PROGRAM P00_OP
VAR		
	N_OP_CMD AT%MB64:  ARRAY [0..35] OF BYTE;//op cmd 주소
	memSetResult: UDINT;	
	b_Test: BOOL;
END_VAR
VAR // added by the converter: edge detectors and wires of the graphical bodies
    _rt1, _rt2, _rt3, _rt4, _rt5, _rt6, _rt7, _rt8, _rt9, _rt10, _rt11, _rt12, _rt13, _rt14, _rt15, _rt16, _rt17, _rt18, _rt19, _rt20, _rt21, _rt22, _rt23, _rt24, _rt25, _rt26, _rt27, _rt28, _rt29, _rt30, _rt31, _rt32, _rt33, _rt34, _rt35, _rt36, _rt37, _rt38, _rt39, _rt40, _rt41, _rt42, _rt43, _rt44, _rt45, _rt46, _rt47, _rt48, _rt49, _rt50, _rt51, _rt52, _rt53, _rt54, _rt55, _rt56, _rt57, _rt58, _rt59, _rt60, _rt61, _rt62, _rt63, _rt64, _rt65, _rt66, _rt67, _rt68, _rt69, _rt70, _rt71, _rt72, _rt73, _rt74, _rt75, _rt76, _rt77, _rt78, _rt79, _rt80, _rt81, _rt82, _rt83, _rt84, _rt85, _rt86, _rt87, _rt88, _rt89, _rt90, _rt91, _rt92, _rt93, _rt94, _rt95, _rt96, _rt97, _rt98, _rt99, _rt100, _rt101, _rt102, _rt103, _rt104, _rt105, _rt106, _rt107, _rt108, _rt109, _rt110, _rt111, _rt112, _rt113, _rt114, _rt115, _rt116, _rt117, _rt118, _rt119, _rt120, _rt121, _rt122, _rt123, _rt124, _rt125, _rt126, _rt127, _rt128, _rt129, _rt130, _rt131, _rt132, _rt133, _rt134, _rt135, _rt136, _rt137, _rt138, _rt139, _rt140, _rt141, _rt142, _rt143, _rt144, _rt145, _rt146, _rt147, _rt148, _rt149, _rt150, _rt151, _rt152, _rt153, _rt154, _rt155, _rt156, _rt157, _rt158, _rt159, _rt160, _rt161, _rt162, _rt163, _rt164, _rt165, _rt166, _rt167, _rt168, _rt169, _rt170, _rt171, _rt172, _rt173, _rt174, _rt175, _rt176, _rt177, _rt178, _rt179, _rt180, _rt181, _rt182, _rt183, _rt184, _rt185, _rt186, _rt187, _rt188, _rt189, _rt190, _rt191, _rt192, _rt193, _rt194, _rt195, _rt196, _rt197, _rt198, _rt199, _rt200, _rt201, _rt202, _rt203, _rt204, _rt205, _rt206, _rt207, _rt208, _rt209, _rt210, _rt211, _rt212, _rt213, _rt214, _rt215, _rt216, _rt217, _rt218, _rt219, _rt220, _rt221, _rt222, _rt223, _rt224, _rt225, _rt226, _rt227, _rt228, _rt229, _rt230, _rt231, _rt232, _rt233, _rt234 : R_TRIG;
    _w1, _w2, _w3, _w4, _w5, _w6, _w7, _w8, _w9, _w10, _w11, _w12 : BOOL;
END_VAR

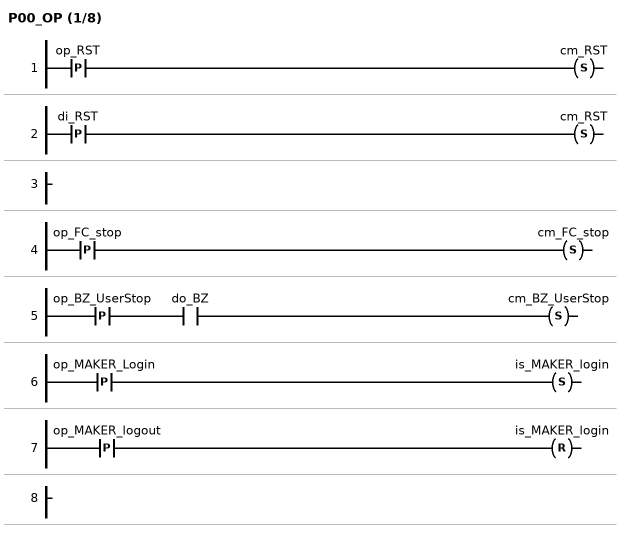
// NETWORK 1
_rt1(CLK := op_RST);
cm_RST S= _rt1.Q;

// NETWORK 2
_rt2(CLK := di_RST);
cm_RST S= _rt2.Q;

// NETWORK 3

// NETWORK 4
_rt3(CLK := op_FC_stop);
cm_FC_stop S= _rt3.Q;

// NETWORK 5
_rt4(CLK := op_BZ_UserStop);
cm_BZ_UserStop S= _rt4.Q AND do_BZ;

// NETWORK 6
_rt5(CLK := op_MAKER_Login);
is_MAKER_login S= _rt5.Q;

// NETWORK 7
_rt6(CLK := op_MAKER_logout);
is_MAKER_login R= _rt6.Q;

// NETWORK 8

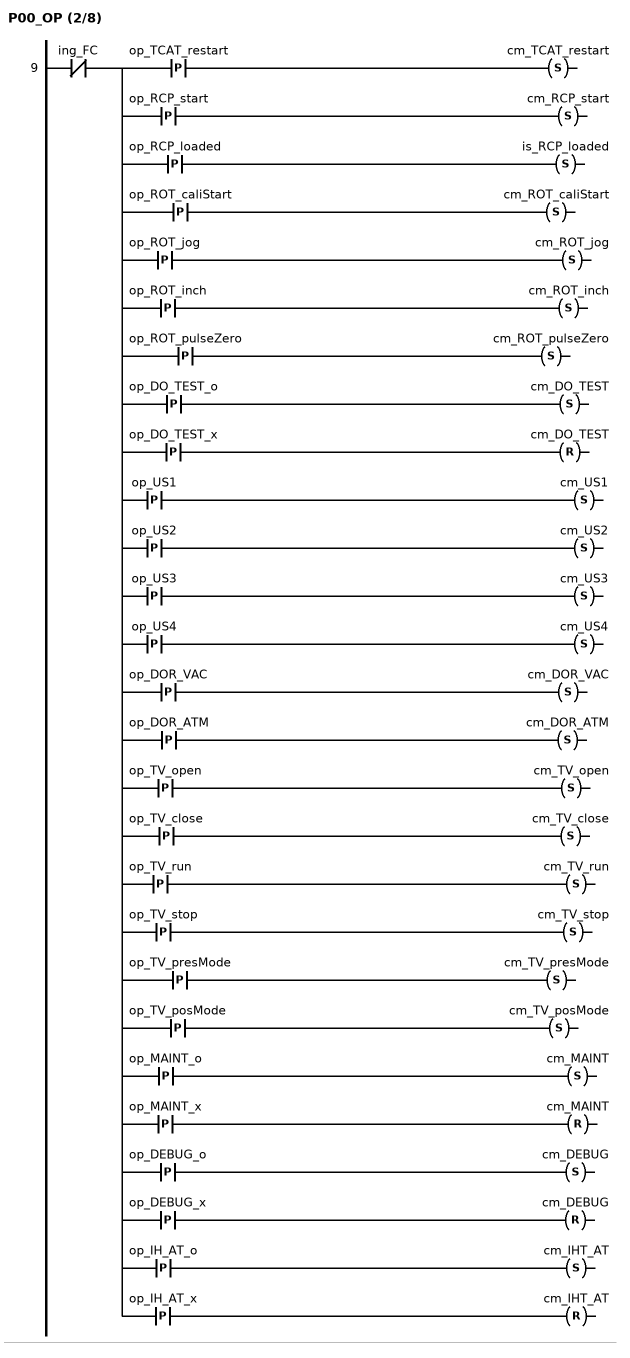
// NETWORK 9
_w1 := NOT ing_FC;
_rt7(CLK := op_TCAT_restart);
cm_TCAT_restart S= _w1 AND _rt7.Q;
_rt8(CLK := op_RCP_start);
cm_RCP_start S= _w1 AND _rt8.Q;
_rt9(CLK := op_RCP_loaded);
is_RCP_loaded S= _w1 AND _rt9.Q;
_rt10(CLK := op_ROT_caliStart);
cm_ROT_caliStart S= _w1 AND _rt10.Q;
_rt11(CLK := op_ROT_jog);
cm_ROT_jog S= _w1 AND _rt11.Q;
_rt12(CLK := op_ROT_inch);
cm_ROT_inch S= _w1 AND _rt12.Q;
_rt13(CLK := op_ROT_pulseZero);
cm_ROT_pulseZero S= _w1 AND _rt13.Q;
_rt14(CLK := op_DO_TEST_o);
cm_DO_TEST S= _w1 AND _rt14.Q;
_rt15(CLK := op_DO_TEST_x);
cm_DO_TEST R= _w1 AND _rt15.Q;
_rt16(CLK := op_US1);
cm_US1 S= _w1 AND _rt16.Q;
_rt17(CLK := op_US2);
cm_US2 S= _w1 AND _rt17.Q;
_rt18(CLK := op_US3);
cm_US3 S= _w1 AND _rt18.Q;
_rt19(CLK := op_US4);
cm_US4 S= _w1 AND _rt19.Q;
_rt20(CLK := op_DOR_VAC);
cm_DOR_VAC S= _w1 AND _rt20.Q;
_rt21(CLK := op_DOR_ATM);
cm_DOR_ATM S= _w1 AND _rt21.Q;
_rt22(CLK := op_TV_open);
cm_TV_open S= _w1 AND _rt22.Q;
_rt23(CLK := op_TV_close);
cm_TV_close S= _w1 AND _rt23.Q;
_rt24(CLK := op_TV_run);
cm_TV_run S= _w1 AND _rt24.Q;
_rt25(CLK := op_TV_stop);
cm_TV_stop S= _w1 AND _rt25.Q;
_rt26(CLK := op_TV_presMode);
cm_TV_presMode S= _w1 AND _rt26.Q;
_rt27(CLK := op_TV_posMode);
cm_TV_posMode S= _w1 AND _rt27.Q;
_rt28(CLK := op_MAINT_o);
cm_MAINT S= _w1 AND _rt28.Q;
_rt29(CLK := op_MAINT_x);
cm_MAINT R= _w1 AND _rt29.Q;
_rt30(CLK := op_DEBUG_o);
cm_DEBUG S= _w1 AND _rt30.Q;
_rt31(CLK := op_DEBUG_x);
cm_DEBUG R= _w1 AND _rt31.Q;
_rt32(CLK := op_IH_AT_o);
cm_IHT_AT S= _w1 AND _rt32.Q;
_rt33(CLK := op_IH_AT_x);
cm_IHT_AT R= _w1 AND _rt33.Q;

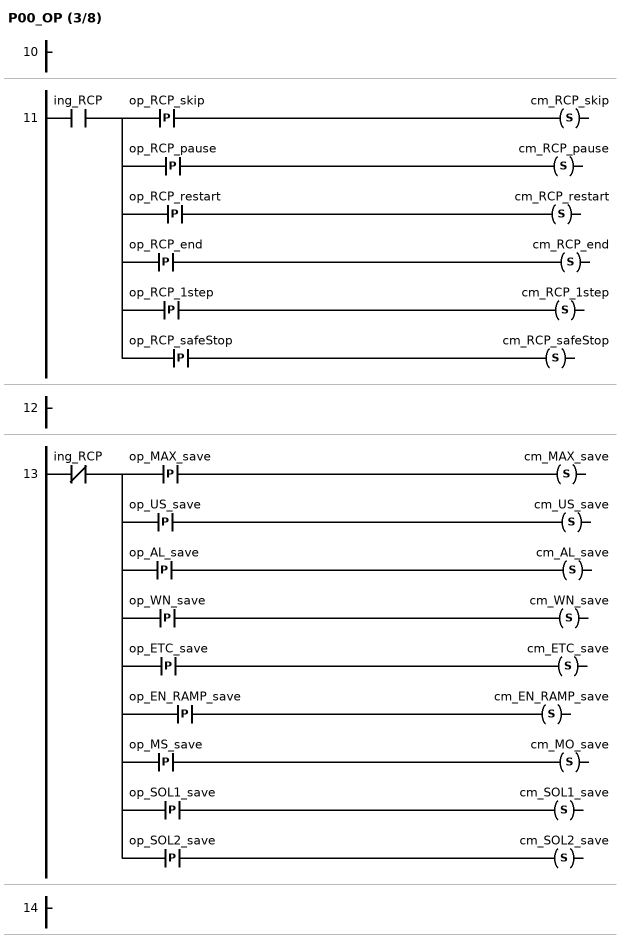
// NETWORK 10

// NETWORK 11
_rt34(CLK := op_RCP_skip);
cm_RCP_skip S= ing_RCP AND _rt34.Q;
_rt35(CLK := op_RCP_pause);
cm_RCP_pause S= ing_RCP AND _rt35.Q;
_rt36(CLK := op_RCP_restart);
cm_RCP_restart S= ing_RCP AND _rt36.Q;
_rt37(CLK := op_RCP_end);
cm_RCP_end S= ing_RCP AND _rt37.Q;
_rt38(CLK := op_RCP_1step);
cm_RCP_1step S= ing_RCP AND _rt38.Q;
_rt39(CLK := op_RCP_safeStop);
cm_RCP_safeStop S= ing_RCP AND _rt39.Q;

// NETWORK 12

// NETWORK 13
_w2 := NOT ing_RCP;
_rt40(CLK := op_MAX_save);
cm_MAX_save S= _w2 AND _rt40.Q;
_rt41(CLK := op_US_save);
cm_US_save S= _w2 AND _rt41.Q;
_rt42(CLK := op_AL_save);
cm_AL_save S= _w2 AND _rt42.Q;
_rt43(CLK := op_WN_save);
cm_WN_save S= _w2 AND _rt43.Q;
_rt44(CLK := op_ETC_save);
cm_ETC_save S= _w2 AND _rt44.Q;
_rt45(CLK := op_EN_RAMP_save);
cm_EN_RAMP_save S= _w2 AND _rt45.Q;
_rt46(CLK := op_MS_save);
cm_MO_save S= _w2 AND _rt46.Q;
_rt47(CLK := op_SOL1_save);
cm_SOL1_save S= _w2 AND _rt47.Q;
_rt48(CLK := op_SOL2_save);
cm_SOL2_save S= _w2 AND _rt48.Q;

// NETWORK 14

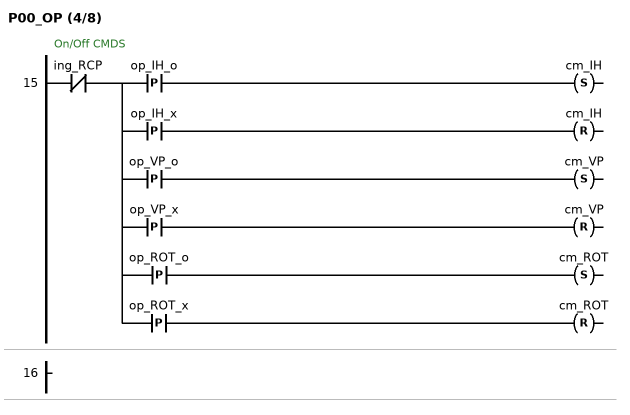
// NETWORK 15
// On/Off CMDS
_w3 := NOT ing_RCP;
_rt49(CLK := op_IH_o);
cm_IH S= _w3 AND _rt49.Q;
_rt50(CLK := op_IH_x);
cm_IH R= _w3 AND _rt50.Q;
_rt51(CLK := op_VP_o);
cm_VP S= _w3 AND _rt51.Q;
_rt52(CLK := op_VP_x);
cm_VP R= _w3 AND _rt52.Q;
_rt53(CLK := op_ROT_o);
cm_ROT S= _w3 AND _rt53.Q;
_rt54(CLK := op_ROT_x);
cm_ROT R= _w3 AND _rt54.Q;

// NETWORK 16

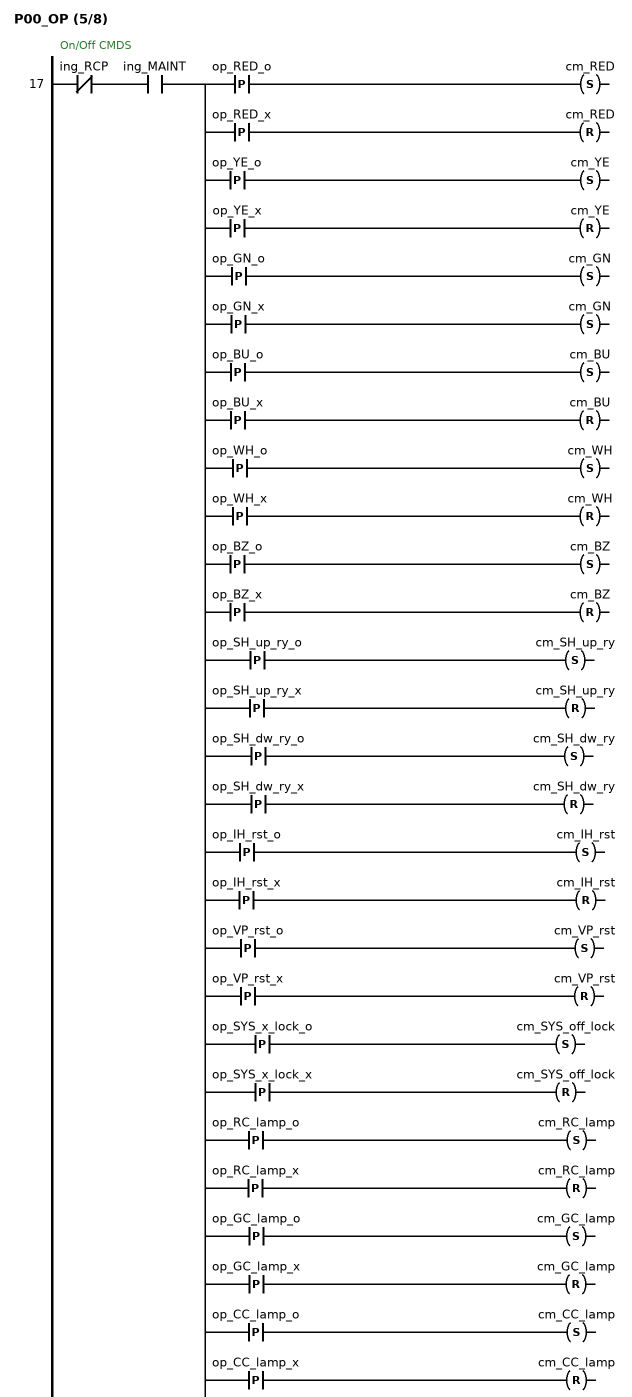
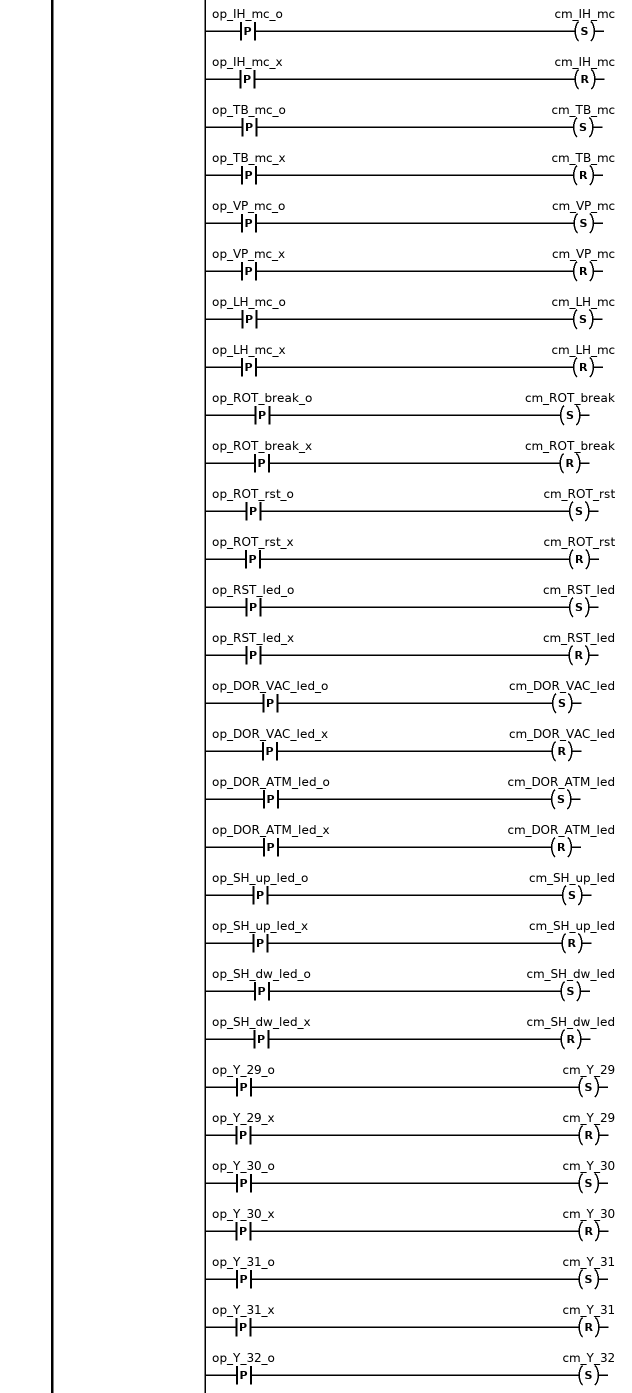
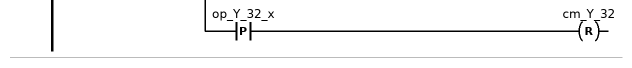
// NETWORK 17
// On/Off CMDS
_w4 := NOT ing_RCP AND ing_MAINT;
_rt55(CLK := op_RED_o);
cm_RED S= _w4 AND _rt55.Q;
_rt56(CLK := op_RED_x);
cm_RED R= _w4 AND _rt56.Q;
_rt57(CLK := op_YE_o);
cm_YE S= _w4 AND _rt57.Q;
_rt58(CLK := op_YE_x);
cm_YE R= _w4 AND _rt58.Q;
_rt59(CLK := op_GN_o);
cm_GN S= _w4 AND _rt59.Q;
_rt60(CLK := op_GN_x);
cm_GN S= _w4 AND _rt60.Q;
_rt61(CLK := op_BU_o);
cm_BU S= _w4 AND _rt61.Q;
_rt62(CLK := op_BU_x);
cm_BU R= _w4 AND _rt62.Q;
_rt63(CLK := op_WH_o);
cm_WH S= _w4 AND _rt63.Q;
_rt64(CLK := op_WH_x);
cm_WH R= _w4 AND _rt64.Q;
_rt65(CLK := op_BZ_o);
cm_BZ S= _w4 AND _rt65.Q;
_rt66(CLK := op_BZ_x);
cm_BZ R= _w4 AND _rt66.Q;
_rt67(CLK := op_SH_up_ry_o);
cm_SH_up_ry S= _w4 AND _rt67.Q;
_rt68(CLK := op_SH_up_ry_x);
cm_SH_up_ry R= _w4 AND _rt68.Q;
_rt69(CLK := op_SH_dw_ry_o);
cm_SH_dw_ry S= _w4 AND _rt69.Q;
_rt70(CLK := op_SH_dw_ry_x);
cm_SH_dw_ry R= _w4 AND _rt70.Q;
_rt71(CLK := op_IH_rst_o);
cm_IH_rst S= _w4 AND _rt71.Q;
_rt72(CLK := op_IH_rst_x);
cm_IH_rst R= _w4 AND _rt72.Q;
_rt73(CLK := op_VP_rst_o);
cm_VP_rst S= _w4 AND _rt73.Q;
_rt74(CLK := op_VP_rst_x);
cm_VP_rst R= _w4 AND _rt74.Q;
_rt75(CLK := op_SYS_x_lock_o);
cm_SYS_off_lock S= _w4 AND _rt75.Q;
_rt76(CLK := op_SYS_x_lock_x);
cm_SYS_off_lock R= _w4 AND _rt76.Q;
_rt77(CLK := op_RC_lamp_o);
cm_RC_lamp S= _w4 AND _rt77.Q;
_rt78(CLK := op_RC_lamp_x);
cm_RC_lamp R= _w4 AND _rt78.Q;
_rt79(CLK := op_GC_lamp_o);
cm_GC_lamp S= _w4 AND _rt79.Q;
_rt80(CLK := op_GC_lamp_x);
cm_GC_lamp R= _w4 AND _rt80.Q;
_rt81(CLK := op_CC_lamp_o);
cm_CC_lamp S= _w4 AND _rt81.Q;
_rt82(CLK := op_CC_lamp_x);
cm_CC_lamp R= _w4 AND _rt82.Q;
_rt83(CLK := op_IH_mc_o);
cm_IH_mc S= _w4 AND _rt83.Q;
_rt84(CLK := op_IH_mc_x);
cm_IH_mc R= _w4 AND _rt84.Q;
_rt85(CLK := op_TB_mc_o);
cm_TB_mc S= _w4 AND _rt85.Q;
_rt86(CLK := op_TB_mc_x);
cm_TB_mc R= _w4 AND _rt86.Q;
_rt87(CLK := op_VP_mc_o);
cm_VP_mc S= _w4 AND _rt87.Q;
_rt88(CLK := op_VP_mc_x);
cm_VP_mc R= _w4 AND _rt88.Q;
_rt89(CLK := op_LH_mc_o);
cm_LH_mc S= _w4 AND _rt89.Q;
_rt90(CLK := op_LH_mc_x);
cm_LH_mc R= _w4 AND _rt90.Q;
_rt91(CLK := op_ROT_break_o);
cm_ROT_break S= _w4 AND _rt91.Q;
_rt92(CLK := op_ROT_break_x);
cm_ROT_break R= _w4 AND _rt92.Q;
_rt93(CLK := op_ROT_rst_o);
cm_ROT_rst S= _w4 AND _rt93.Q;
_rt94(CLK := op_ROT_rst_x);
cm_ROT_rst R= _w4 AND _rt94.Q;
_rt95(CLK := op_RST_led_o);
cm_RST_led S= _w4 AND _rt95.Q;
_rt96(CLK := op_RST_led_x);
cm_RST_led R= _w4 AND _rt96.Q;
_rt97(CLK := op_DOR_VAC_led_o);
cm_DOR_VAC_led S= _w4 AND _rt97.Q;
_rt98(CLK := op_DOR_VAC_led_x);
cm_DOR_VAC_led R= _w4 AND _rt98.Q;
_rt99(CLK := op_DOR_ATM_led_o);
cm_DOR_ATM_led S= _w4 AND _rt99.Q;
_rt100(CLK := op_DOR_ATM_led_x);
cm_DOR_ATM_led R= _w4 AND _rt100.Q;
_rt101(CLK := op_SH_up_led_o);
cm_SH_up_led S= _w4 AND _rt101.Q;
_rt102(CLK := op_SH_up_led_x);
cm_SH_up_led R= _w4 AND _rt102.Q;
_rt103(CLK := op_SH_dw_led_o);
cm_SH_dw_led S= _w4 AND _rt103.Q;
_rt104(CLK := op_SH_dw_led_x);
cm_SH_dw_led R= _w4 AND _rt104.Q;
_rt105(CLK := op_Y_29_o);
cm_Y_29 S= _w4 AND _rt105.Q;
_rt106(CLK := op_Y_29_x);
cm_Y_29 R= _w4 AND _rt106.Q;
_rt107(CLK := op_Y_30_o);
cm_Y_30 S= _w4 AND _rt107.Q;
_rt108(CLK := op_Y_30_x);
cm_Y_30 R= _w4 AND _rt108.Q;
_rt109(CLK := op_Y_31_o);
cm_Y_31 S= _w4 AND _rt109.Q;
_rt110(CLK := op_Y_31_x);
cm_Y_31 R= _w4 AND _rt110.Q;
_rt111(CLK := op_Y_32_o);
cm_Y_32 S= _w4 AND _rt111.Q;
_rt112(CLK := op_Y_32_x);
cm_Y_32 R= _w4 AND _rt112.Q;

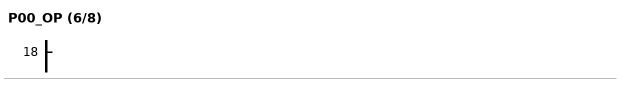
// NETWORK 18

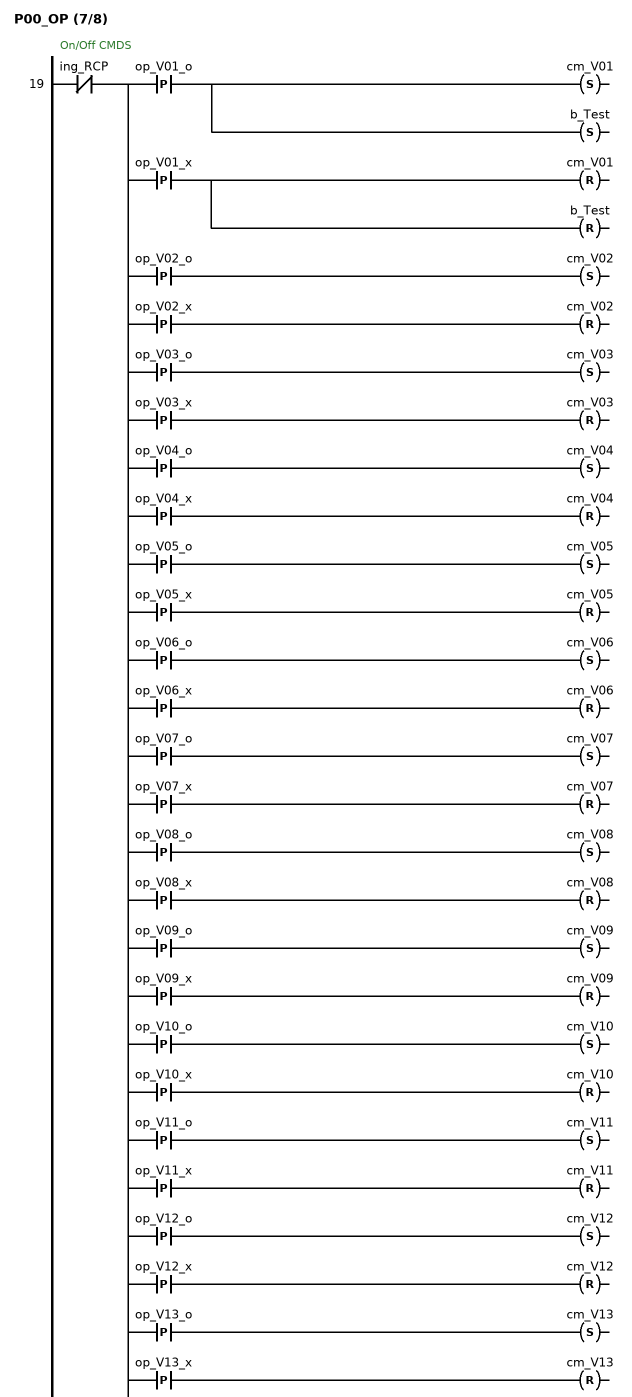
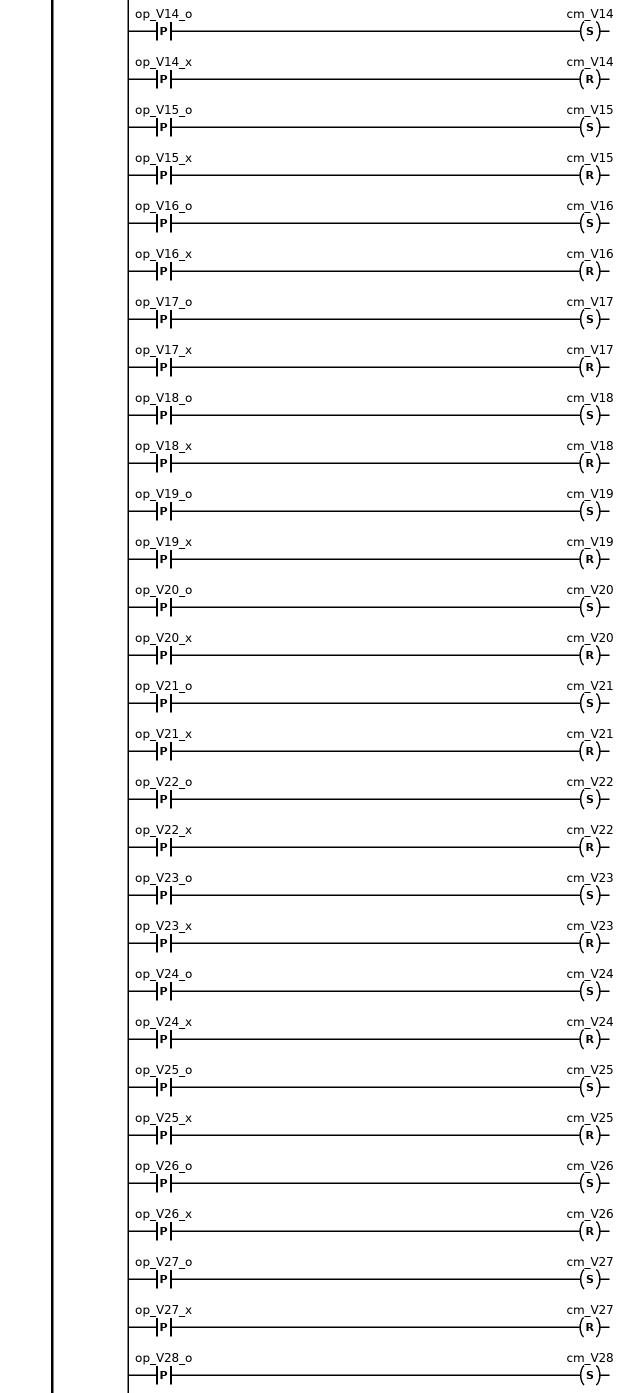
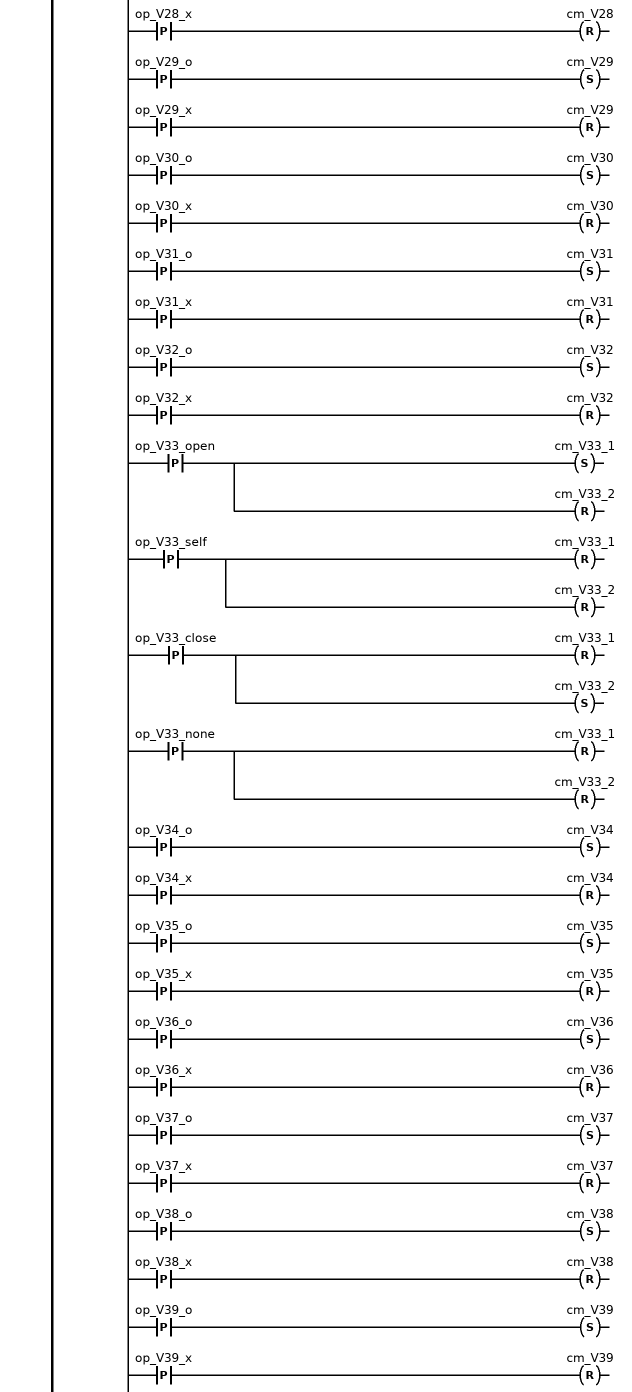
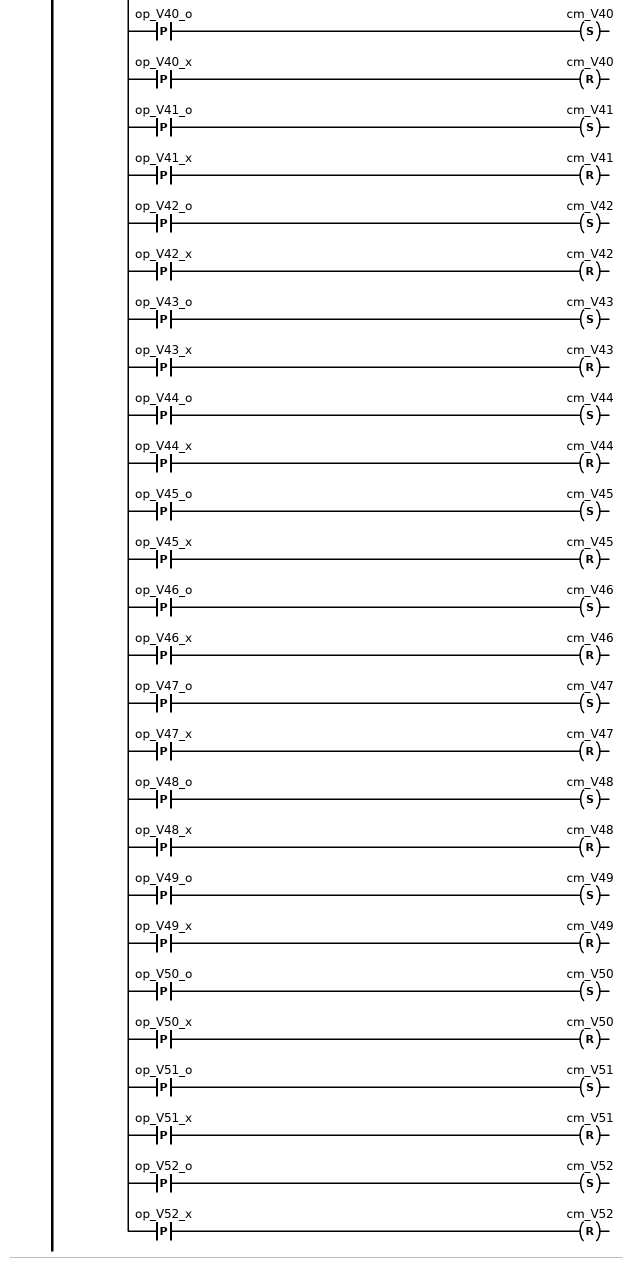
// NETWORK 19
// On/Off CMDS
_w5 := NOT ing_RCP;
_rt113(CLK := op_V01_o);
_w6 := _w5 AND _rt113.Q;
cm_V01 S= _w6;
b_Test S= _w6;
_rt114(CLK := op_V01_x);
_w7 := _w5 AND _rt114.Q;
cm_V01 R= _w7;
b_Test R= _w7;
_rt115(CLK := op_V02_o);
cm_V02 S= _w5 AND _rt115.Q;
_rt116(CLK := op_V02_x);
cm_V02 R= _w5 AND _rt116.Q;
_rt117(CLK := op_V03_o);
cm_V03 S= _w5 AND _rt117.Q;
_rt118(CLK := op_V03_x);
cm_V03 R= _w5 AND _rt118.Q;
_rt119(CLK := op_V04_o);
cm_V04 S= _w5 AND _rt119.Q;
_rt120(CLK := op_V04_x);
cm_V04 R= _w5 AND _rt120.Q;
_rt121(CLK := op_V05_o);
cm_V05 S= _w5 AND _rt121.Q;
_rt122(CLK := op_V05_x);
cm_V05 R= _w5 AND _rt122.Q;
_rt123(CLK := op_V06_o);
cm_V06 S= _w5 AND _rt123.Q;
_rt124(CLK := op_V06_x);
cm_V06 R= _w5 AND _rt124.Q;
_rt125(CLK := op_V07_o);
cm_V07 S= _w5 AND _rt125.Q;
_rt126(CLK := op_V07_x);
cm_V07 R= _w5 AND _rt126.Q;
_rt127(CLK := op_V08_o);
cm_V08 S= _w5 AND _rt127.Q;
_rt128(CLK := op_V08_x);
cm_V08 R= _w5 AND _rt128.Q;
_rt129(CLK := op_V09_o);
cm_V09 S= _w5 AND _rt129.Q;
_rt130(CLK := op_V09_x);
cm_V09 R= _w5 AND _rt130.Q;
_rt131(CLK := op_V10_o);
cm_V10 S= _w5 AND _rt131.Q;
_rt132(CLK := op_V10_x);
cm_V10 R= _w5 AND _rt132.Q;
_rt133(CLK := op_V11_o);
cm_V11 S= _w5 AND _rt133.Q;
_rt134(CLK := op_V11_x);
cm_V11 R= _w5 AND _rt134.Q;
_rt135(CLK := op_V12_o);
cm_V12 S= _w5 AND _rt135.Q;
_rt136(CLK := op_V12_x);
cm_V12 R= _w5 AND _rt136.Q;
_rt137(CLK := op_V13_o);
cm_V13 S= _w5 AND _rt137.Q;
_rt138(CLK := op_V13_x);
cm_V13 R= _w5 AND _rt138.Q;
_rt139(CLK := op_V14_o);
cm_V14 S= _w5 AND _rt139.Q;
_rt140(CLK := op_V14_x);
cm_V14 R= _w5 AND _rt140.Q;
_rt141(CLK := op_V15_o);
cm_V15 S= _w5 AND _rt141.Q;
_rt142(CLK := op_V15_x);
cm_V15 R= _w5 AND _rt142.Q;
_rt143(CLK := op_V16_o);
cm_V16 S= _w5 AND _rt143.Q;
_rt144(CLK := op_V16_x);
cm_V16 R= _w5 AND _rt144.Q;
_rt145(CLK := op_V17_o);
cm_V17 S= _w5 AND _rt145.Q;
_rt146(CLK := op_V17_x);
cm_V17 R= _w5 AND _rt146.Q;
_rt147(CLK := op_V18_o);
cm_V18 S= _w5 AND _rt147.Q;
_rt148(CLK := op_V18_x);
cm_V18 R= _w5 AND _rt148.Q;
_rt149(CLK := op_V19_o);
cm_V19 S= _w5 AND _rt149.Q;
_rt150(CLK := op_V19_x);
cm_V19 R= _w5 AND _rt150.Q;
_rt151(CLK := op_V20_o);
cm_V20 S= _w5 AND _rt151.Q;
_rt152(CLK := op_V20_x);
cm_V20 R= _w5 AND _rt152.Q;
_rt153(CLK := op_V21_o);
cm_V21 S= _w5 AND _rt153.Q;
_rt154(CLK := op_V21_x);
cm_V21 R= _w5 AND _rt154.Q;
_rt155(CLK := op_V22_o);
cm_V22 S= _w5 AND _rt155.Q;
_rt156(CLK := op_V22_x);
cm_V22 R= _w5 AND _rt156.Q;
_rt157(CLK := op_V23_o);
cm_V23 S= _w5 AND _rt157.Q;
_rt158(CLK := op_V23_x);
cm_V23 R= _w5 AND _rt158.Q;
_rt159(CLK := op_V24_o);
cm_V24 S= _w5 AND _rt159.Q;
_rt160(CLK := op_V24_x);
cm_V24 R= _w5 AND _rt160.Q;
_rt161(CLK := op_V25_o);
cm_V25 S= _w5 AND _rt161.Q;
_rt162(CLK := op_V25_x);
cm_V25 R= _w5 AND _rt162.Q;
_rt163(CLK := op_V26_o);
cm_V26 S= _w5 AND _rt163.Q;
_rt164(CLK := op_V26_x);
cm_V26 R= _w5 AND _rt164.Q;
_rt165(CLK := op_V27_o);
cm_V27 S= _w5 AND _rt165.Q;
_rt166(CLK := op_V27_x);
cm_V27 R= _w5 AND _rt166.Q;
_rt167(CLK := op_V28_o);
cm_V28 S= _w5 AND _rt167.Q;
_rt168(CLK := op_V28_x);
cm_V28 R= _w5 AND _rt168.Q;
_rt169(CLK := op_V29_o);
cm_V29 S= _w5 AND _rt169.Q;
_rt170(CLK := op_V29_x);
cm_V29 R= _w5 AND _rt170.Q;
_rt171(CLK := op_V30_o);
cm_V30 S= _w5 AND _rt171.Q;
_rt172(CLK := op_V30_x);
cm_V30 R= _w5 AND _rt172.Q;
_rt173(CLK := op_V31_o);
cm_V31 S= _w5 AND _rt173.Q;
_rt174(CLK := op_V31_x);
cm_V31 R= _w5 AND _rt174.Q;
_rt175(CLK := op_V32_o);
cm_V32 S= _w5 AND _rt175.Q;
_rt176(CLK := op_V32_x);
cm_V32 R= _w5 AND _rt176.Q;
_rt177(CLK := op_V33_open);
_w8 := _w5 AND _rt177.Q;
cm_V33_1 S= _w8;
cm_V33_2 R= _w8;
_rt178(CLK := op_V33_self);
_w9 := _w5 AND _rt178.Q;
cm_V33_1 R= _w9;
cm_V33_2 R= _w9;
_rt179(CLK := op_V33_close);
_w10 := _w5 AND _rt179.Q;
cm_V33_1 R= _w10;
cm_V33_2 S= _w10;
_rt180(CLK := op_V33_none);
_w11 := _w5 AND _rt180.Q;
cm_V33_1 R= _w11;
cm_V33_2 R= _w11;
_rt181(CLK := op_V34_o);
cm_V34 S= _w5 AND _rt181.Q;
_rt182(CLK := op_V34_x);
cm_V34 R= _w5 AND _rt182.Q;
_rt183(CLK := op_V35_o);
cm_V35 S= _w5 AND _rt183.Q;
_rt184(CLK := op_V35_x);
cm_V35 R= _w5 AND _rt184.Q;
_rt185(CLK := op_V36_o);
cm_V36 S= _w5 AND _rt185.Q;
_rt186(CLK := op_V36_x);
cm_V36 R= _w5 AND _rt186.Q;
_rt187(CLK := op_V37_o);
cm_V37 S= _w5 AND _rt187.Q;
_rt188(CLK := op_V37_x);
cm_V37 R= _w5 AND _rt188.Q;
_rt189(CLK := op_V38_o);
cm_V38 S= _w5 AND _rt189.Q;
_rt190(CLK := op_V38_x);
cm_V38 R= _w5 AND _rt190.Q;
_rt191(CLK := op_V39_o);
cm_V39 S= _w5 AND _rt191.Q;
_rt192(CLK := op_V39_x);
cm_V39 R= _w5 AND _rt192.Q;
_rt193(CLK := op_V40_o);
cm_V40 S= _w5 AND _rt193.Q;
_rt194(CLK := op_V40_x);
cm_V40 R= _w5 AND _rt194.Q;
_rt195(CLK := op_V41_o);
cm_V41 S= _w5 AND _rt195.Q;
_rt196(CLK := op_V41_x);
cm_V41 R= _w5 AND _rt196.Q;
_rt197(CLK := op_V42_o);
cm_V42 S= _w5 AND _rt197.Q;
_rt198(CLK := op_V42_x);
cm_V42 R= _w5 AND _rt198.Q;
_rt199(CLK := op_V43_o);
cm_V43 S= _w5 AND _rt199.Q;
_rt200(CLK := op_V43_x);
cm_V43 R= _w5 AND _rt200.Q;
_rt201(CLK := op_V44_o);
cm_V44 S= _w5 AND _rt201.Q;
_rt202(CLK := op_V44_x);
cm_V44 R= _w5 AND _rt202.Q;
_rt203(CLK := op_V45_o);
cm_V45 S= _w5 AND _rt203.Q;
_rt204(CLK := op_V45_x);
cm_V45 R= _w5 AND _rt204.Q;
_rt205(CLK := op_V46_o);
cm_V46 S= _w5 AND _rt205.Q;
_rt206(CLK := op_V46_x);
cm_V46 R= _w5 AND _rt206.Q;
_rt207(CLK := op_V47_o);
cm_V47 S= _w5 AND _rt207.Q;
_rt208(CLK := op_V47_x);
cm_V47 R= _w5 AND _rt208.Q;
_rt209(CLK := op_V48_o);
cm_V48 S= _w5 AND _rt209.Q;
_rt210(CLK := op_V48_x);
cm_V48 R= _w5 AND _rt210.Q;
_rt211(CLK := op_V49_o);
cm_V49 S= _w5 AND _rt211.Q;
_rt212(CLK := op_V49_x);
cm_V49 R= _w5 AND _rt212.Q;
_rt213(CLK := op_V50_o);
cm_V50 S= _w5 AND _rt213.Q;
_rt214(CLK := op_V50_x);
cm_V50 R= _w5 AND _rt214.Q;
_rt215(CLK := op_V51_o);
cm_V51 S= _w5 AND _rt215.Q;
_rt216(CLK := op_V51_x);
cm_V51 R= _w5 AND _rt216.Q;
_rt217(CLK := op_V52_o);
cm_V52 S= _w5 AND _rt217.Q;
_rt218(CLK := op_V52_x);
cm_V52 R= _w5 AND _rt218.Q;

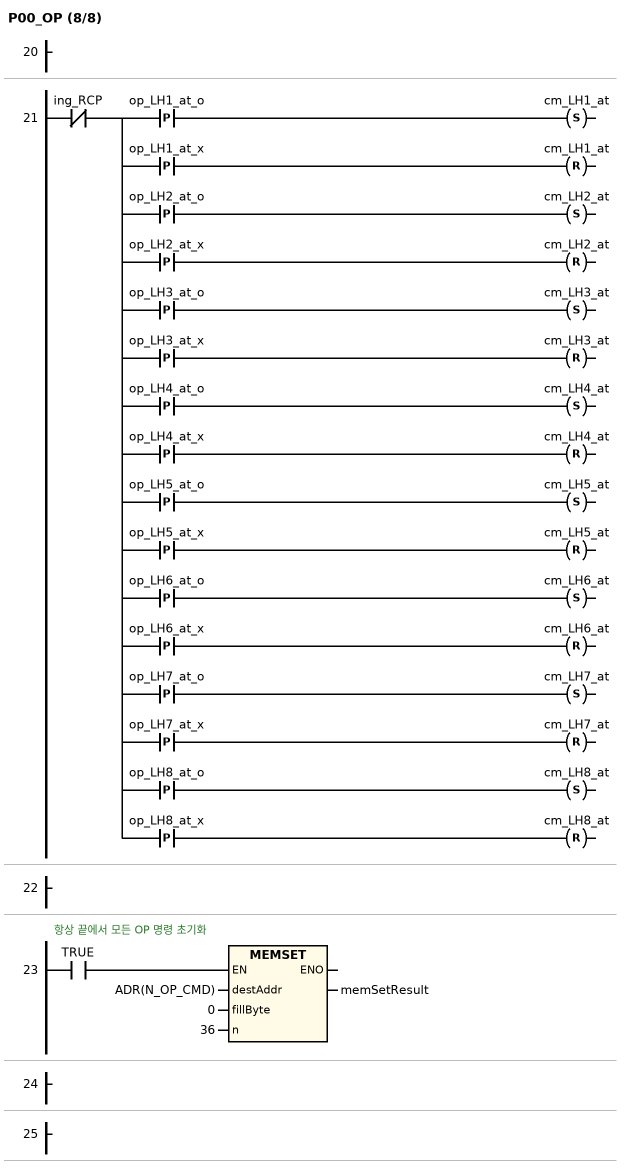
// NETWORK 20

// NETWORK 21
_w12 := NOT ing_RCP;
_rt219(CLK := op_LH1_at_o);
cm_LH1_at S= _w12 AND _rt219.Q;
_rt220(CLK := op_LH1_at_x);
cm_LH1_at R= _w12 AND _rt220.Q;
_rt221(CLK := op_LH2_at_o);
cm_LH2_at S= _w12 AND _rt221.Q;
_rt222(CLK := op_LH2_at_x);
cm_LH2_at R= _w12 AND _rt222.Q;
_rt223(CLK := op_LH3_at_o);
cm_LH3_at S= _w12 AND _rt223.Q;
_rt224(CLK := op_LH3_at_x);
cm_LH3_at R= _w12 AND _rt224.Q;
_rt225(CLK := op_LH4_at_o);
cm_LH4_at S= _w12 AND _rt225.Q;
_rt226(CLK := op_LH4_at_x);
cm_LH4_at R= _w12 AND _rt226.Q;
_rt227(CLK := op_LH5_at_o);
cm_LH5_at S= _w12 AND _rt227.Q;
_rt228(CLK := op_LH5_at_x);
cm_LH5_at R= _w12 AND _rt228.Q;
_rt229(CLK := op_LH6_at_o);
cm_LH6_at S= _w12 AND _rt229.Q;
_rt230(CLK := op_LH6_at_x);
cm_LH6_at R= _w12 AND _rt230.Q;
_rt231(CLK := op_LH7_at_o);
cm_LH7_at S= _w12 AND _rt231.Q;
_rt232(CLK := op_LH7_at_x);
cm_LH7_at R= _w12 AND _rt232.Q;
_rt233(CLK := op_LH8_at_o);
cm_LH8_at S= _w12 AND _rt233.Q;
_rt234(CLK := op_LH8_at_x);
cm_LH8_at R= _w12 AND _rt234.Q;

// NETWORK 22

// NETWORK 23
// 항상 끝에서 모든 OP 명령 초기화
memSetResult := MEMSET(destAddr := ADR(N_OP_CMD), fillByte := 0, n := 36);

// NETWORK 24

// NETWORK 25

END_PROGRAM

(* stored: Version 1.1.0.1, ProductVersion 3.1.4024.12
   POU P00_OP: Id {a4953bcd-8e5b-444a-83cf-7140b289623a}, SpecialFunc None *)
